FUNCTION_BLOCK PUBL_132_BOTTOM_AND_SIDE_ROUGH_MILLING-PLANAR_FACE-SIMPLE (* 132-variable local group publisher for milling a planar_face *)
  (* Standard: 61499-2 *)
  (* Version 1.0, 21-03-12, GASR, Universidade do Estado de Santa Catarina *)
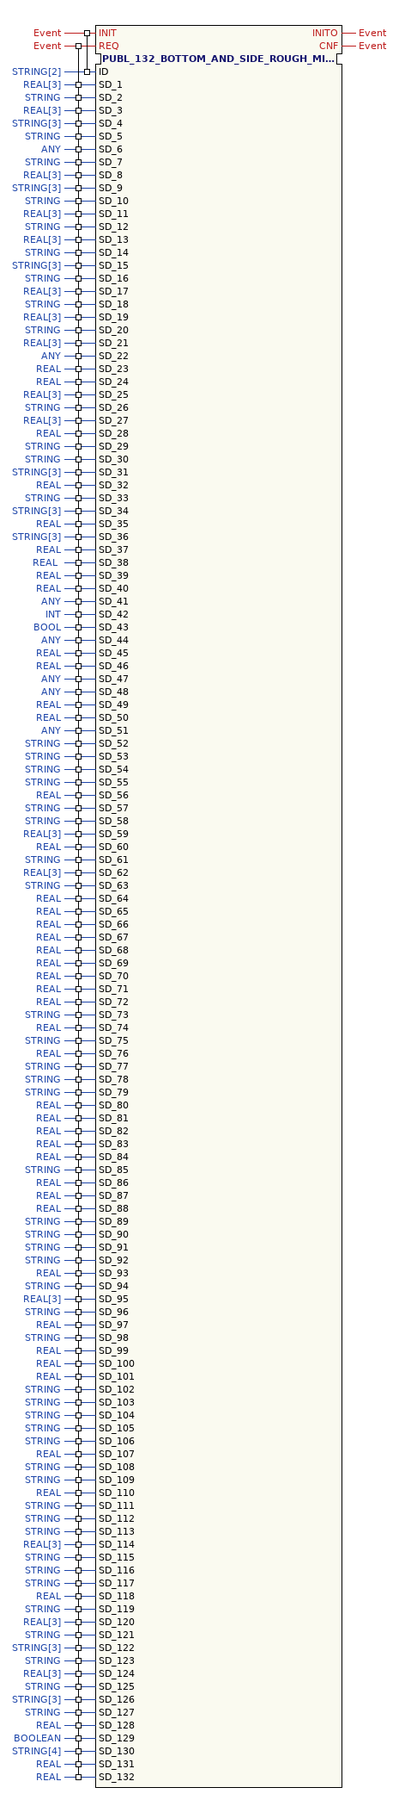
  EVENT_INPUT
    INIT WITH ID; (* Service Initialization *)
    REQ WITH SD_1, SD_2, SD_3, SD_4, SD_5, SD_6, SD_7, SD_8, SD_9, SD_10, SD_11, SD_12, SD_13, SD_14, SD_15, SD_16, SD_17, SD_18, SD_19, SD_20, SD_21, SD_22, SD_23, SD_24, SD_25, SD_26, SD_27, SD_28, SD_29, SD_30, SD_31, SD_32, SD_33, SD_34, SD_35, SD_36, SD_37, SD_38, SD_39, SD_40, SD_41, SD_42, SD_43, SD_44, SD_45, SD_46, SD_47, SD_48, SD_49, SD_50, SD_51, SD_52, SD_53, SD_54, SD_55, SD_56, SD_57, SD_58, SD_59, SD_60, SD_61, SD_62, SD_63, SD_64, SD_65, SD_66, SD_67, SD_68, SD_69, SD_70, SD_71, SD_72, SD_73, SD_74, SD_75, SD_76, SD_77, SD_78, SD_79, SD_80, SD_81, SD_82, SD_83, SD_84, SD_85, SD_86, SD_87, SD_88, SD_89, SD_90, SD_91, SD_92, SD_93, SD_94, SD_95, SD_96, SD_97, SD_98, SD_99, SD_100, SD_101, SD_102, SD_103, SD_104, SD_105, SD_106, SD_107, SD_108, SD_109, SD_110, SD_111, SD_112, SD_113, SD_114, SD_115, SD_116, SD_117, SD_118, SD_119, SD_120, SD_121, SD_122, SD_123, SD_124, SD_125, SD_126, SD_127, SD_128, SD_129, SD_130, SD_131, SD_132; (* Service Request *)
  END_EVENT
  EVENT_OUTPUT
    INITO; (* Initialization Confirm *)
    CNF; (* Service Confirmation *)
  END_EVENT
  VAR_INPUT
    ID : ARRAY [0..1] OF STRING; (* PLANAR_FACE instance name, SUBL instance name *)
    SD_1 : ARRAY [0..2] OF REAL; (* pos *)
    SD_2 : STRING; (* current_tool *)
    SD_3 : ARRAY [0..2] OF REAL; (* setup.its_secplane.position.location.coordinates *)
    SD_4 : ARRAY [0..2] OF STRING; (* manufacturing_feature.its_id *)
    SD_5 : STRING; (* manufacturing_feature.its_workpiece.its_id *)
    SD_6 : ANY; (* manufacturing_feature.its_operations *)
    SD_7 : STRING; (* two5d_manufacturing_feature.Feature_placement.Name *)
    SD_8 : ARRAY [0..2] OF REAL; (* two5d_manufacturing_feature.Feature_placement.Location.Coordinates *)
    SD_9 : ARRAY [0..2] OF STRING; (* two5d_manufacturing_feature.Feature_placement.Location.Name *)
    SD_10 : STRING; (* two5d_manufacturing_feature.Feature_placement.OP Axis.its_id *)
    SD_11 : ARRAY [0..2] OF REAL; (* two5d_manufacturing_feature.Feature_placement.OP Axis.Direction_ratios *)
    SD_12 : STRING; (* two5d_manufacturing_feature.Feature_placement.OP Ref_direction.its_id *)
    SD_13 : ARRAY [0..2] OF REAL; (* two5d_manufacturing_feature.Feature_placement.OP Ref_direction.Direction_ratios *)
    SD_14 : STRING; (* machining_feature.Depth.Name *)
    SD_15 : ARRAY [0..2] OF STRING; (* machining_feature.Depth.Position.Name *)
    SD_16 : STRING; (* machining_feature.Depth.Position.Location.Name *)
    SD_17 : ARRAY [0..2] OF REAL; (* machining_feature.Depth.Position.Location.Coordinates *)
    SD_18 : STRING; (* machining_feature.Depth.Position.OP Axis.its_id *)
    SD_19 : ARRAY [0..2] OF REAL; (* machining_feature.Depth.Position.OP Axis.Direction_ratios *)
    SD_20 : STRING; (* machining_feature.Depth.Position.OP Ref_direction.its_id *)
    SD_21 : ARRAY [0..2] OF REAL; (* machining_feature.Depth.Position.OP Ref_direction.Direction_ratios *)
    SD_22 : ANY; (* Planar_Face.Course_of_Travel.Distance *)
    SD_23 : REAL; (* Planar_Face.Course_of_Travel.Distance.Theoretical_Size *)
    SD_24 : REAL; (* Planar_Face.Course_of_Travel.Distance.Implicit_Tolerance *)
    SD_25 : ARRAY [0..2] OF REAL; (* Planar_Face.Course_of_Travel.Distance.{vector} = {upper_limit, lower_limit, significant_digits} or {deviation, grade, its_fitting_type} *)
    SD_26 : STRING; (* Planar_Face.Course_of_Travel.Its_Direction.Its_Id *)
    SD_27 : ARRAY [0..2] OF REAL; (* Planar_Face.Course_of_Travel.Its_Direction.Direction_Ratios *)
    SD_28 : REAL; (* Planar_Face.Removal_Boundary.Profile_Length.Its_Parameter_Value *)
    SD_29 : STRING; (* Planar_Face.Removal_Boundary.Profile_Length.Its_Parameter_Unit *)
    SD_30 : STRING; (* Planar_Face.Face_Boundary *)
    SD_31 : ARRAY [0..2] OF STRING; (* Planar_Face.Face_Boundary.Placement.Name *)
    SD_32 : REAL; (* Planar_Face.Face_Boundary.Placement.Location.Coordinates *)
    SD_33 : STRING; (* Planar_Face.Face_Boundary.Placement.Location.Name *)
    SD_34 : ARRAY [0..2] OF STRING; (* Planar_Face.Face_Boundary.Placement.OP Axis.its_id *)
    SD_35 : REAL; (* Planar_Face.Face_Boundary.Placement.OP Axis.Direction_Ratios *)
    SD_36 : ARRAY [0..2] OF STRING; (* Planar_Face.Face_Boundary.Placement.OP Ref_Direction.its_id *)
    SD_37 : REAL; (* Planar_Face.Face_Boundary.Placement.OP Ref_Direction.Direction_ratios *)
    SD_38 : REAL ; (* Planar_Face.Face_Boundary.Diameter *)
    SD_39 : REAL; (* Planar_Face.Face_Boundary.Diameter.Theoretical_Size *)
    SD_40 : REAL; (* Planar_Face.Face_Boundary.Diameter.Implicit_Tolerance *)
    SD_41 : ANY; (* Planar_Face.Face_Boundary.Diameter.{vector} = {upper_limit, lower_limit, significant_digits} or {deviation, grade, its_fitting_type} *)
    SD_42 : INT; (* Planar_Face.Face_Boundary.Number_of_Sides *)
    SD_43 : BOOL; (* Planar_Face.Face_Boundary.Circumscribed_or_Across_Flats *)
    SD_44 : ANY; (* Planar_Face.Face_Boundary.Profile_Width *)
    SD_45 : REAL; (* Planar_Face.Face_Boundary.Profile_Width.Theoretical_Size *)
    SD_46 : REAL; (* Planar_Face.Face_Boundary.Profile_Width.Implicit_Tolerance *)
    SD_47 : ANY; (* Planar_Face.Face_Boundary.Profile_Width.{vector} = {upper_limit, lower_limit, significant_digits} or {deviation, grade, its_fitting_type} *)
    SD_48 : ANY; (* Planar_Face.Face_Boundary.Profile_Length *)
    SD_49 : REAL; (* Planar_Face.Face_Boundary.Profile_Length.Theoretical_Size *)
    SD_50 : REAL; (* Planar_Face.Face_Boundary.Profile_Width.Length_Tolerance *)
    SD_51 : ANY; (* Planar_Face.Face_Boundary.Profile_Length.{vector} = {upper_limit, lower_limit, significant_digits} or {deviation, grade, its_fitting_type} *)
    SD_52 : STRING; (* Planar_Face.Its_Boss.its_id *)
    SD_53 : STRING; (* Planar_Face.Face_Boundary.General_Closed_Profile *)
    SD_54 : STRING; (* Planar_Face.Face_Boundary.Closed_Profile_Shape.Name *)
    SD_55 : STRING; (* Planar_Face.Face_Boundary.Closed_Profile_Shape.Points.Name *)
    SD_56 : REAL; (* Planar_Face.Face_Boundary.Closed_Profile_Shape.Points.Coordinates *)
    SD_57 : STRING; (* bottom_and_side_rough_milling.its_id *)
    SD_58 : STRING; (* its_toolpath.its_list *)
    SD_59 : ARRAY [0..2] OF REAL; (* its_tool_direction *)
    SD_60 : REAL; (* retract_plane *)
    SD_61 : STRING; (* start_point.name *)
    SD_62 : ARRAY [0..2] OF REAL; (* start_point.coordinates *)
    SD_63 : STRING; (* its_tool.its_id *)
    SD_64 : REAL; (* its_tool.its_tool_body.dimension.diameter *)
    SD_65 : REAL; (* its_tool.its_tool_body.dimension.tool_tip_half_angle *)
    SD_66 : REAL; (* its_tool.its_tool_body.dimension.tool_circumference_angle *)
    SD_67 : REAL; (* its_tool.its_tool_body.dimension.cutting_edge_lenght *)
    SD_68 : REAL; (* its_tool.its_tool_body.dimension.edge_radius *)
    SD_69 : REAL; (* its_tool.its_tool_body.dimension.edge_center_vertical *)
    SD_70 : REAL; (* its_tool.its_tool_body.dimension.edge_center_horizontal *)
    SD_71 : REAL; (* its_tool.its_tool_body.number_of_teeth *)
    SD_72 : REAL; (* its_tool.its_tool_body.hand_of_cut *)
    SD_73 : STRING; (* its_tool.its_tool_body.coolant_through *)
    SD_74 : REAL; (* its_tool.its_tool_body.pilot_length *)
    SD_75 : STRING; (* its_tool.its_tool_body.{other_tool_body_parameter} *)
    SD_76 : REAL; (* its_tool.its_cutting_edge.tool_offset_length *)
    SD_77 : STRING; (* its_tool.its_cutting_edge.its_material.standard_identifier *)
    SD_78 : STRING; (* its_tool.its_cutting_edge.its_material.material_identifier *)
    SD_79 : STRING; (* its_tool.its_cutting_edge.its_material.material_property.{list_of_parameters} *)
    SD_80 : REAL; (* its_tool.its_cutting_edge.its_technological_data.cutting_angle *)
    SD_81 : REAL; (* its_tool.its_cutting_edge.its_technological_data.free_angle *)
    SD_82 : REAL; (* its_tool.its_cutting_edge.its_technological_data.aux_angle *)
    SD_83 : REAL; (* its_tool.its_cutting_edge.expected_tool_life *)
    SD_84 : REAL; (* its_tool.its_cutting_edge.its_technology.feedrate *)
    SD_85 : STRING; (* its_tool.its_cutting_edge.its_technology.feedrate_reference *)
    SD_86 : REAL; (* its_tool.its_cutting_edge.its_technology.cutspeed *)
    SD_87 : REAL; (* its_tool.its_cutting_edge.its_technology.spindle *)
    SD_88 : REAL; (* its_tool.its_cutting_edge.its_technology.feedrate_per_tooth *)
    SD_89 : STRING; (* its_tool.its_cutting_edge.its_technology.sincronize_spindle_with_feed *)
    SD_90 : STRING; (* its_tool.its_cutting_edge.its_technology.inhibit_feedrate_override *)
    SD_91 : STRING; (* its_tool.its_cutting_edge.its_technology.inhibit_spindle_override *)
    SD_92 : STRING; (* its_tool.its_cutting_edge.its_technology.its_adaptive_control *)
    SD_93 : REAL; (* its_tool.overall_assembly_length *)
    SD_94 : STRING; (* its_tool.direction_for_spindle_orientation.its_id *)
    SD_95 : ARRAY [0..2] OF REAL; (* its_tool.direction_for_spindle_orientation.direction_ratios *)
    SD_96 : STRING; (* its_tool.tool_holder_diameter_for_spindle_orientation *)
    SD_97 : REAL; (* its_technology.feedrate *)
    SD_98 : STRING; (* its_technology.feedrate_reference *)
    SD_99 : REAL; (* its_technology.cutspeed *)
    SD_100 : REAL; (* its_technology.spindle *)
    SD_101 : REAL; (* its_technology.feedrate_per_tooth *)
    SD_102 : STRING; (* its_technology.sincronize_spindle_with_feed *)
    SD_103 : STRING; (* its_technology.inhibit_feedrate_override *)
    SD_104 : STRING; (* its_technology.inhibit_spindle_override *)
    SD_105 : STRING; (* its_technology.its_adaptive_control *)
    SD_106 : STRING; (* its_machine_functions.coolant *)
    SD_107 : REAL; (* its_machine_functions.coolant_pressure *)
    SD_108 : STRING; (* its_machine_functions.mist *)
    SD_109 : STRING; (* its_machine_functions.through_spindle_coolant *)
    SD_110 : REAL; (* its_machine_functions.through_pressure *)
    SD_111 : STRING; (* its_machine_functions.axis_clamping *)
    SD_112 : STRING; (* its_machine_functions.chip_removal *)
    SD_113 : STRING; (* its_machine_functions.oriented_spindle_stop.its_id *)
    SD_114 : ARRAY [0..2] OF REAL; (* its_machine_functions.oriented_spindle_stop.direction_ratios *)
    SD_115 : STRING; (* its_machine_functions.its_process_model.ini_data_file *)
    SD_116 : STRING; (* its_machine_functions.its_process_model.its_type *)
    SD_117 : STRING; (* its_machine_functions.other_functions *)
    SD_118 : REAL; (* overcut_length *)
    SD_119 : STRING; (* approach.tool_orientation.its_id *)
    SD_120 : ARRAY [0..2] OF REAL; (* approach.tool_orientation.direction_ratios *)
    SD_121 : STRING; (* approach.approach_retract_strategy (name of it) *)
    SD_122 : ARRAY [0..2] OF STRING; (* approach.approach_retract_strategy.list of parameters *)
    SD_123 : STRING; (* retract.tool_orientation.its_id *)
    SD_124 : ARRAY [0..2] OF REAL; (* retract.tool_orientation.direction_ratios *)
    SD_125 : STRING; (* retract.approach_retract_strategy (name of it) *)
    SD_126 : ARRAY [0..2] OF STRING; (* retract.approach_retract_strategy.list of parameters *)
    SD_127 : STRING; (* its_machining_strategy *)
    SD_128 : REAL; (* its_machining_strategy.overlap *)
    SD_129 : BOOLEAN; (* its_machining_strategy.allow_multiple_passes *)
    SD_130 : ARRAY [0..3] OF STRING; (* its_machining_strategy.list of parameters *)
    SD_131 : REAL; (* axial_cutting_depth *)
    SD_132 : REAL; (* allowance_bottom *)
  END_VAR
  SERVICE PUBL_132/SUBL_132 (* Data publication service *)
    SEQUENCE normal_establishment
      PUBL_132.INIT(ID) -> SUBL_132.INITO();
      SUBL_132.INIT(ID) -> SUBL_132.INITO();
    END_SEQUENCE
    SEQUENCE normal_data_transfer
      PUBL_132.REQ(SD_1,SD_2,SD_3,SD_4,SD_5,SD_6,SD_7,SD_8,SD_9,SD_10,SD_11,SD_12,SD_13,SD_14,SD_15,SD_16,SD_17,SD_18,SD_19,SD_20,SD_21,SD_22,SD_23,SD_24,SD_25,SD_26,SD_27,SD_28,SD_29,SD_30,SD_31,SD_32,SD_33,SD_34,SD_35,SD_36,SD_37,SD_38,SD_39,SD_40,SD_41,SD_42,SD_43,SD_44,SD_45,SD_46,SD_47,SD_48,SD_49,SD_50,SD_51,SD_52,SD_53,SD_54,SD_55,SD_56,SD_57,SD_58,SD_59,SD_60,SD_61,SD_62,SD_63,SD_64,SD_65,SD_66,SD_67,SD_68,SD_69,SD_70,SD_71,SD_72,SD_73,SD_74,SD_75,SD_76,SD_77,SD_78,SD_79,SD_80,SD_81,SD_82,SD_83,SD_84,SD_85,SD_86,SD_87,SD_88,SD_89,SD_90,SD_91,SD_92,SD_93,SD_94,SD_95,SD_96,SD_97,SD_98,SD_99,SD_100,SD_101,SD_102,SD_103,SD_104,SD_105,SD_106,SD_107,SD_108,SD_109,SD_110,SD_111,SD_112,SD_113,SD_114,SD_115,SD_116,SD_117,SD_118,SD_119,SD_120,SD_121,SD_122,SD_123,SD_124,SD_125,SD_126,SD_127,SD_128,SD_129,SD_130,SD_131,SD_132) -> SUBL_132.IND(RD_1,RD_2,RD_3,RD_4,RD_5,RD_6,RD_7,RD_8,RD_9,RD_10,RD_11,RD_12,RD_13,RD_14,RD_15,RD_16,RD_17,RD_18,RD_19,RD_20,RD_21,RD_22,RD_23,RD_24,RD_25,RD_26,RD_27,RD_28,RD_29,RD_30,RD_31,RD_32,RD_33,RD_34,RD_35,RD_36,RD_37,RD_38,RD_39,RD_40,RD_41,RD_42,RD_43,RD_44,RD_45,RD_46,RD_47,RD_48,RD_49,RD_50,RD_51,RD_52,RD_53,RD_54,RD_55,RD_56,RD_57,RD_58,RD_59,RD_60,RD_61,RD_62,RD_63,RD_64,RD_65,RD_66,RD_67,RD_68,RD_69,RD_70,RD_71,RD_72,RD_73,RD_74,RD_75,RD_76,RD_77,RD_78,RD_79,RD_80,RD_81,RD_82,RD_83,RD_84,RD_85,RD_86,RD_87,RD_88,RD_89,RD_90,RD_91,RD_92,RD_93,RD_94,RD_95,RD_96,RD_97,RD_98,RD_99,RD_100,RD_101,RD_102,RD_103,RD_104,RD_105,RD_106,RD_107,RD_108,RD_109,RD_110,RD_111,RD_112,RD_113,RD_114,RD_115,RD_116,RD_117,RD_118,RD_119,RD_120,RD_121,RD_122,RD_123,RD_124,RD_125,RD_126,RD_127,RD_128,RD_129,RD_130,RD_131,RD_132);
    END_SEQUENCE
  END_SERVICE
END_FUNCTION_BLOCK
